FUNCTION_BLOCK FB_CondensingBoiler
VAR_INPUT
END_VAR
VAR_OUTPUT
END_VAR
VAR
END_VAR

END_FUNCTION_BLOCK

(* stored: Version 1.1.0.1, ProductVersion 3.1.4024.10
   POU FB_CondensingBoiler: Id {a735ace5-71e9-497d-839f-87ce45582673}, SpecialFunc None *)
